FUNCTION_BLOCK FB_Element IMPLEMENTS I_Material
(*
Intended to represent an element and some associated state values with that element.
Allows external access to overwrite properties of the element.
If a property is set to an invalid value, and the name of the element can be found
in the property lookup table, then the invalid value is overwritten to the value
found in the lookup table.
If a property is set to an invalid value and the provided element name is not found
in the property lookup table, the value is left as is and the error boolean is set
and an error message is set.
If a property is set to a valid value, even if the value disagrees with the value
found in that property's lookup table, then the value is left as in regardless
of the validity of the element name currently set.
Values that are not properties are not intended to be written to or read directly.
Always use the properties to interface with the function block.
*)
VAR
    {attribute 'pytmc' := '
        pv: Mass
        io: io
    '}
    fMass : LREAL;

    {attribute 'pytmc' := '
        pv: Name
        io: io
    '}
    sName : STRING;

    {attribute 'pytmc' := '
        pv: Protons
        io: io
    '}
    nProtons : INT;

    {attribute 'pytmc' := '
        pv: Density
        io: io
    '}
    fDensity : LREAL;

    {attribute 'pytmc' := '
        pv: Error
        io: i
    '}
    bError : BOOL;

    {attribute 'pytmc' := '
        pv: ErrorMsg
        io: i
    '}
    sErrorMsg : T_MaxString;
END_VAR


PROPERTY Density : LREAL
GET

DensityCheck(fDensityIn := fDensity);

Density := fDensity;
END_GET
SET

DensityCheck(fDensityIn := Density);

fDensity := Density;
END_SET
END_PROPERTY


METHOD DensityCheck : BOOL
VAR_IN_OUT
    fDensityIn : LREAL;
END_VAR
VAR
    fbElementDensity : FB_ElementDensity;
END_VAR

// If we have an invalid density value, try to look it up in the element density lookup table.
IF fDensityIn <= 0.0 THEN
    // Use lookup table to get the density for the specified name.
    fbElementDensity(
        sName := Name,
        bFound =>,
        fValue =>
    );
    // If we find the name in the lookup table, update the density.
    IF fbElementDensity.bFound THEN
        fDensity := fbElementDensity.fValue;
        DensityCheck := TRUE;
    ELSE
        // Set the error bit true if we still have an invalid density.
        bError := TRUE;
        sErrorMsg := CONCAT('Invalid density value of: [',
            CONCAT(LREAL_TO_STRING(fDensity),
            CONCAT(']. Unable to find element named: [',
            CONCAT(Name,
            '] in the lookup table.'))));
        DensityCheck := FALSE;
    END_IF
ELSE
    DensityCheck := TRUE;
END_IF
END_METHOD


PROPERTY Error : BOOL
GET

bError := FALSE;
sErrorMsg := '';

fMass := Mass;
sName := Name;
nProtons := Protons;
fDensity := Density;

Error := bError;
END_GET
END_PROPERTY

PROPERTY ErrorMsg : T_MaxString
GET

bError := Error;

ErrorMsg := sErrorMsg;
END_GET
END_PROPERTY


PROPERTY Mass : LREAL
GET

MassCheck(fMassIn := fMass);

Mass := fMass;
END_GET
SET

MassCheck(fMassIn := Mass);

fMass := Mass;
END_SET
END_PROPERTY


METHOD MassCheck : BOOL
VAR_IN_OUT
    fMassIn : LREAL;
END_VAR
VAR
    fbAtomicMass : FB_AtomicMass;
END_VAR

// If we have an invalid mass value, try to look it up in the atomic mass lookup table.
IF fMass <= 0.0 THEN
    // Use lookup table to get atomic mass for specified name.
    fbAtomicMass(
        sName := Name,
        bFound =>,
        fValue =>
    );
    // If we find the name in the lookup table, update the mass.
    IF fbAtomicMass.bFound THEN
        fMass := fbAtomicMass.fValue;
        MassCheck := TRUE;
    ELSE
        // Set the error bit true if we still have an invalid mass.
        bError := TRUE;
        sErrorMsg := CONCAT('Invalid mass value of: [',
            CONCAT(LREAL_TO_STRING(fMass),
            CONCAT(']. Unable to find element named: [',
            CONCAT(Name,
            '] in the lookup table.'))));
        MassCheck := FALSE;
    END_IF
ELSE
    MassCheck := TRUE;
END_IF
END_METHOD


PROPERTY Name : STRING
GET

Name := sName;
END_GET
SET

sName := Name;
END_SET
END_PROPERTY


PROPERTY Protons : INT
GET

ProtonsCheck(nProtonsIn := nProtons);

Protons := nProtons;
END_GET
SET

ProtonsCheck(nProtonsIn := Protons);

nProtons := Protons;
END_SET
END_PROPERTY


METHOD ProtonsCheck : BOOL
VAR_IN_OUT
    nProtonsIn : INT;
END_VAR
VAR
    fbAtomicNumber : FB_AtomicNumber;
END_VAR

// If we have an invalid number of protons value, try to look it up in the atomic number lookup table.
IF nProtonsIn <= 0 THEN
    // Use lookup table to get number of protons for specified element name.
    fbAtomicNumber(
        sName := Name,
        bFound =>,
        nValue =>
    );
    // If we find the name in the lookup table, update the number of protons.
    IF fbAtomicNumber.bFound THEN
        nProtons := fbAtomicNumber.nValue;
        ProtonsCheck := TRUE;
    ELSE
        // Set the error bit true if we still have an invalid number of protons.
        bError := TRUE;
        sErrorMsg := CONCAT('Invalid number of protons: [',
            CONCAT(INT_TO_STRING(nProtons),
            CONCAT(']. Unable to find element named: [',
            CONCAT(Name,
            '] in the lookup table.'))));
        ProtonsCheck := FALSE;
    END_IF
ELSE
    ProtonsCheck := TRUE;
END_IF
END_METHOD


METHOD SetState
VAR_INPUT
    fMass : LREAL;
    sName : STRING;
    nProtons : INT;
    fDensity : LREAL;
END_VAR

Name := sName;
Mass := fMass;
Protons := nProtons;
Density := fDensity;

//bError := Error;
END_METHOD

END_FUNCTION_BLOCK

(* stored: Version 1.1.0.1, ProductVersion 3.1.4022.18
   POU FB_Element: Id {036736e7-f9bf-4a69-9445-0ffc36020f10}, SpecialFunc None
   Property Density: Id {5988db1c-263a-49f3-827c-d3d591debf39}
   Get Get: Id {9a40a13c-c07c-49e4-a85c-18c7660f376b}
   Set Set: Id {03c2386c-b342-4210-a3ed-0752fc2f7a47}
   Method DensityCheck: Id {56e3f75e-c0d8-4d00-a79a-a9f9becb722c}
   Property Error: Id {60f55223-0106-4252-ac7a-fa8496e5b982}
   Get Get: Id {cb0a7a02-656b-432b-97f0-4183d73bda25}
   Property ErrorMsg: Id {8dc270f2-9dde-4384-b6b1-af8e5748dbe9}
   Get Get: Id {9bcb73db-a52f-4679-9e83-6a9e0afdd554}
   Property Mass: Id {31b2a0f1-ae0a-4416-ab03-b332ea566adc}
   Get Get: Id {d0cbf8b3-8e2a-4602-a6ac-ca017dd74765}
   Set Set: Id {36480fed-1dda-4006-a1fe-211e4981789a}
   Method MassCheck: Id {abe420d5-f48d-4692-b2e8-d9451205a4ac}
   Property Name: Id {220e42b2-72cf-4b6b-96e0-b36ccb11227c}
   Get Get: Id {f8a8189e-379c-47fd-b4a7-b767e0d98d8c}
   Set Set: Id {80fdff07-2ae3-4fb9-aac3-d0d80b5aa529}
   Property Protons: Id {610ab6d9-b89e-4c2d-b83d-9d312c3f4503}
   Get Get: Id {5197a756-cb36-445b-8219-2749bf1125bd}
   Set Set: Id {e661cef8-a37e-4dbd-87ed-dc44de405e59}
   Method ProtonsCheck: Id {cb6adc19-5d74-4f68-b965-6370a7ad7f74}
   Method SetState: Id {25429d11-6525-4e0f-962f-7c5660e2977e} *)
